// TIA Portal V16 export
// export: Created 2021-07-12T14:47:20.5224601Z, ExportSetting WithDefaults, DisplayName Totally Integrated Automation Portal, DisplayVersion V16, DisplayName TIA Portal Version Control Interface, DisplayVersion V16, DisplayName TIA Portal Openness, DisplayVersion V16, DisplayName STEP 7 Professional, DisplayVersion V16, DisplayName STEP 7 Safety, DisplayVersion V16, DisplayName WinCC Professional, DisplayVersion V16
TYPE "SimaHydTO_typeHMIConnectionGetCharacteristicInterfaceCommand"
TITLE = SimaHydTO_typeHMIConnectionGetCharacteristicInterfaceCommand
// Function block command interface of FB "GetCharacteristics"
// stored: IsFailsafeCompliant false
   STRUCT
      execute : Bool;   // Start measurement
      abort : Bool;   // Stop measurement
      enableRampingForward : Bool := True;   // Enable ramping of Q-Output value (voltage) in positivedirection
      enableRampingBackward : Bool := True;   // Enable ramping of Q-Output value (voltage) in negative direction
      saveConfig : Bool;   // Save measurement configuration
      loadConfig : Bool;   // Load measurement configuration
   END_STRUCT;
END_TYPE
